Fanuc KAREL source: kd00061.KL

-- PROVISIONAL review KL for V940-1; original PC SHA256 8ae64affcb4156ab29b8a235f708ad0f88ee5904540a9e8a6a4c995b123c62a9
-- Incomplete behavior may be omitted. Consult companion uncertainty JSON. Do not deploy.
PROGRAM KD00061
%NOLOCKGROUP
VAR
  I : INTEGER
  J : INTEGER
  B : BOOLEAN
  R : REAL
  S : STRING[80]
BEGIN
  -- V9_ZERO_TABLE_METADATA_HINT layout=0001; no indexed target words; source/name/runtime held
  -- UNRESOLVED_PC offsets 5-18; opcodes 9D,81,18,9D,1B,9D,12,9D,13,04
  -- UNRESOLVED_PC offsets 23-27; opcodes 7F
END KD00061
